% RSLogix 500 project wind.RSS %
PROJECT "WIND"    % processor: SLC 500, 1747-L543 %

PROGRAM FILES
  LAD 2 "MAIN"  12 rungs  %   %
  LAD 3 "AZ MAN CON"  4 rungs
  LAD 4 "AZ PID CON"  7 rungs
  LAD 5 "DATA XFER"  3 rungs
  LAD 6 "ALT MAN C"  4 rungs
  LAD 7 "ALT PID C"  6 rungs

DATA FILES
  O0 OUTPUT  21 elements
  I1 INPUT  21 elements
  S2 STATUS  164 elements
  B3 BINARY  1 elements
  T4 TIMER  1 elements
  C5 COUNTER  1 elements
  R6 CONTROL  1 elements
  N7 INTEGER  30 elements
  F8 FLOAT  1 elements
  N10 AZ PID  30 elements  % PID Control File %
  N11 ALT PID  30 elements

LADDER 2 "MAIN"    %   %
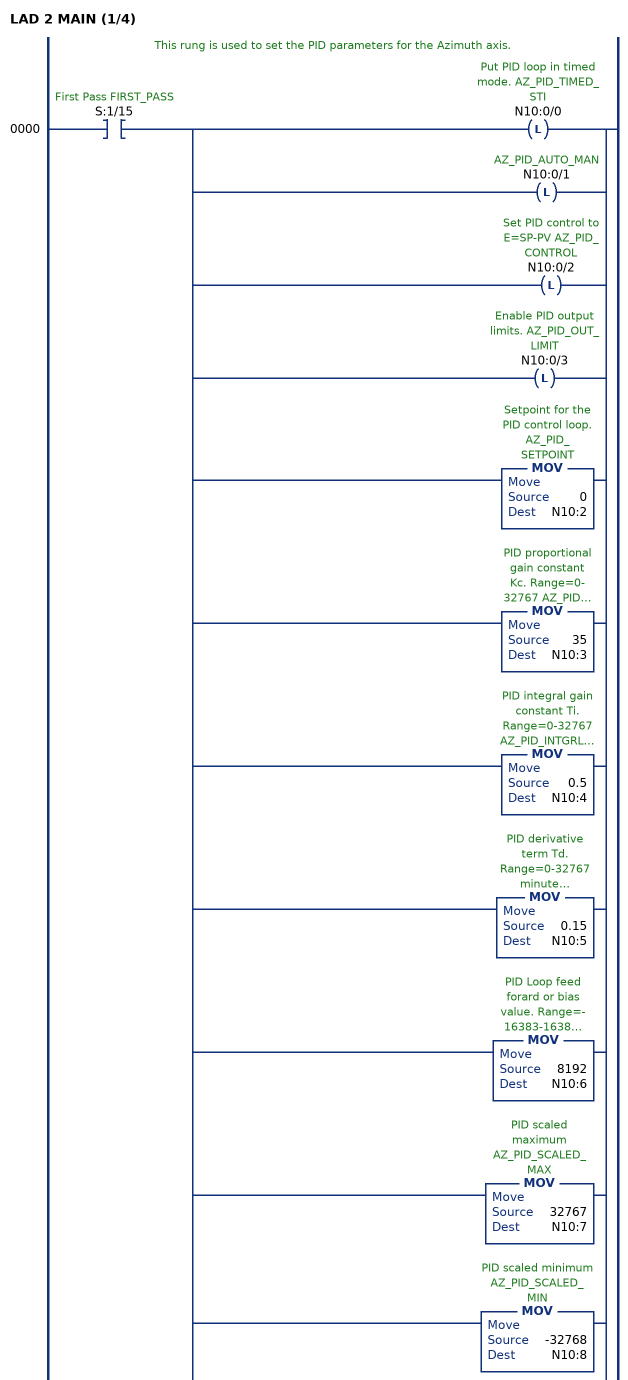
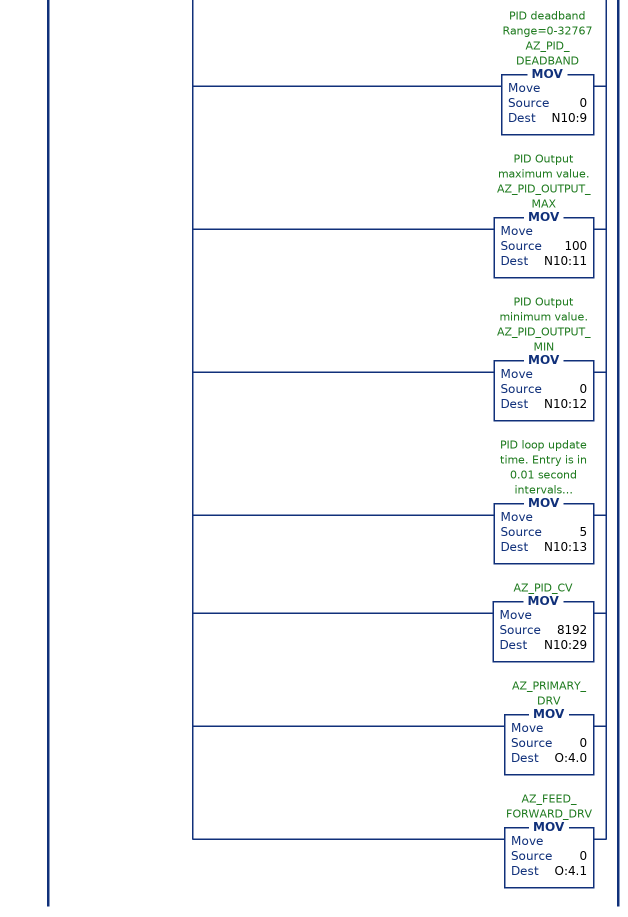
% Rung: 0 %
% This rung is used to set the PID parameters for the Azimuth axis. %
SOR XIC S:1/15 BST OTL N10:0/0 NXB OTL N10:0/1 NXB OTL N10:0/2 NXB OTL N10:0/3 NXB MOV 0 N10:2 NXB MOV 35 N10:3 NXB MOV 0.5 N10:4 NXB MOV 0.15 N10:5 NXB MOV 8192 N10:6 NXB MOV 32767 N10:7 NXB MOV -32768 N10:8 NXB MOV 0 N10:9 NXB MOV 100 N10:11 NXB MOV 0 N10:12 NXB MOV 5 N10:13 NXB MOV 8192 N10:29 NXB MOV 0 O:4.0 NXB MOV 0 O:4.1 BND EOR
%   S:1/15  FIRST_PASS  "First Pass" %
%   N10:0/0  AZ_PID_TIMED_STI  "Put PID loop in timed mode." %
%   N10:0/1  AZ_PID_AUTO_MAN %
%   OTL N10:0/1  "Put PID Loop in Manual Control." %
%   N10:0/2  AZ_PID_CONTROL  "Set PID control to E=SP-PV" %
%   N10:0/3  AZ_PID_OUT_LIMIT  "Enable PID output limits." %
%   N10:2  AZ_PID_SETPOINT  "Setpoint for the PID control loop." %
%   N10:3  AZ_PID_GAIN  "PID proportional gain constant Kc. Range=0-32767" %
%   N10:4  AZ_PID_INTGRL_GAIN  "PID integral gain constant Ti. Range=0-32767" %
%   N10:5  AZ_PID_DER_TERM  "PID derivative term Td. Range=0-32767 minutes" %
%   N10:6  AZ_PID_BIAS  "PID Loop feed forard or bias value. Range=-16383-16383" %
%   N10:7  AZ_PID_SCALED_MAX  "PID scaled maximum" %
%   N10:8  AZ_PID_SCALED_MIN  "PID scaled minimum" %
%   N10:9  AZ_PID_DEADBAND  "PID deadband Range=0-32767" %
%   N10:11  AZ_PID_OUTPUT_MAX  "PID Output maximum value." %
%   N10:12  AZ_PID_OUTPUT_MIN  "PID Output minimum value." %
%   N10:13  AZ_PID_LOOP_UPDATE  "PID loop update time. Entry is in 0.01 second intervals. Range=0.01-10.24 sec" %
%   N10:29  AZ_PID_CV %
%   O:4.0  AZ_PRIMARY_DRV %
%   MOV O:4.0  "Set Az Primary Control Output to zero." %
%   O:4.1  AZ_FEED_FORWARD_DRV %
%   MOV O:4.1  "Set Az feed forward output to zero." %

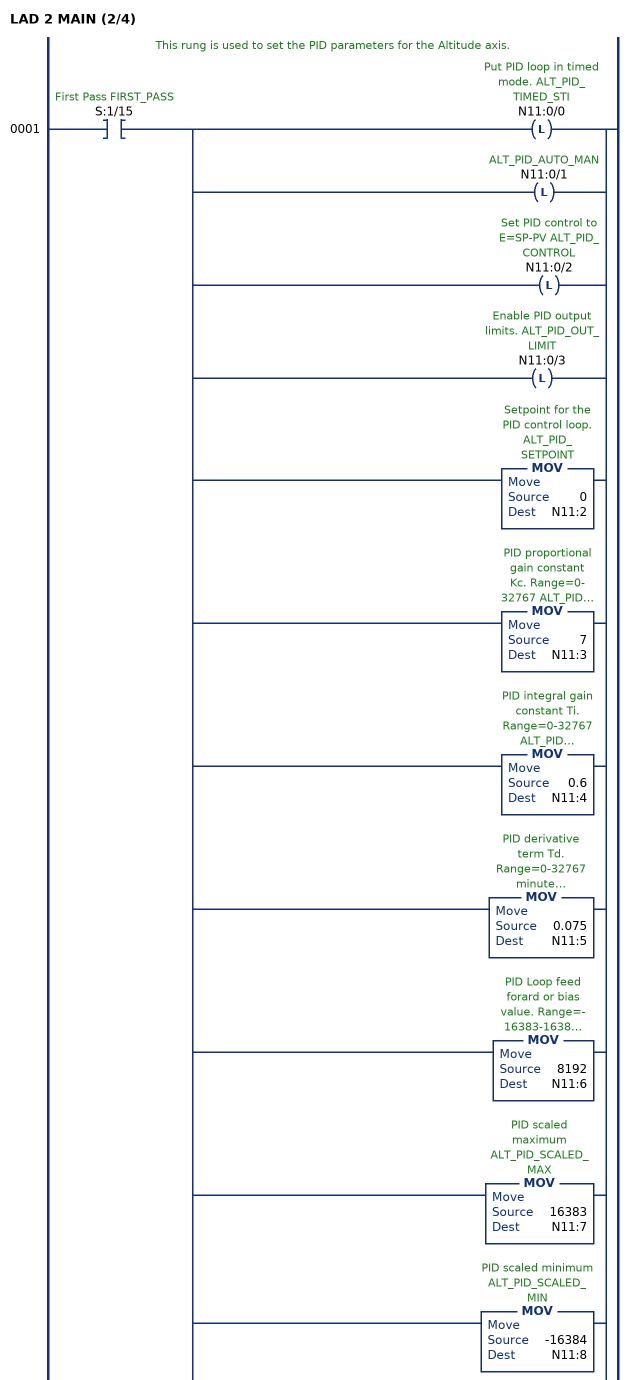

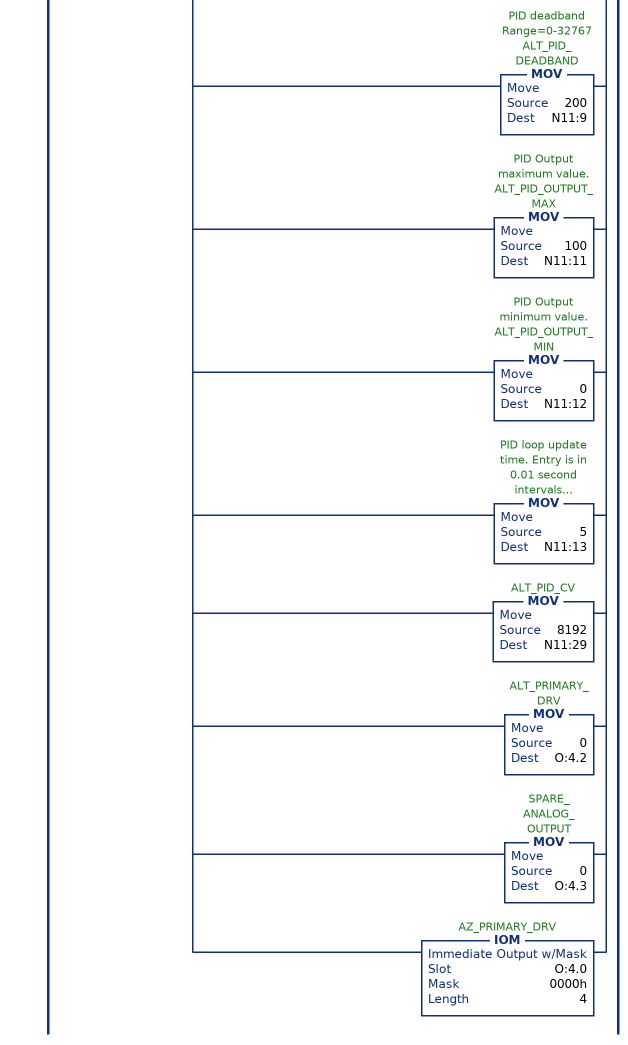
% Rung: 1 %
% This rung is used to set the PID parameters for the Altitude axis. %
SOR XIC S:1/15 BST OTL N11:0/0 NXB OTL N11:0/1 NXB OTL N11:0/2 NXB OTL N11:0/3 NXB MOV 0 N11:2 NXB MOV 7 N11:3 NXB MOV 0.6 N11:4 NXB MOV 0.075 N11:5 NXB MOV 8192 N11:6 NXB MOV 16383 N11:7 NXB MOV -16384 N11:8 NXB MOV 200 N11:9 NXB MOV 100 N11:11 NXB MOV 0 N11:12 NXB MOV 5 N11:13 NXB MOV 8192 N11:29 NXB MOV 0 O:4.2 NXB MOV 0 O:4.3 NXB IOM O:4.0 0000h 4 BND EOR
%   S:1/15  FIRST_PASS  "First Pass" %
%   N11:0/0  ALT_PID_TIMED_STI  "Put PID loop in timed mode." %
%   N11:0/1  ALT_PID_AUTO_MAN %
%   N11:0/2  ALT_PID_CONTROL  "Set PID control to E=SP-PV" %
%   N11:0/3  ALT_PID_OUT_LIMIT  "Enable PID output limits." %
%   N11:2  ALT_PID_SETPOINT  "Setpoint for the PID control loop." %
%   N11:3  ALT_PID_GAIN  "PID proportional gain constant Kc. Range=0-32767" %
%   N11:4  ALT_PID_INTGRL_GAIN  "PID integral gain constant Ti. Range=0-32767" %
%   N11:5  ALT_PID_DER_TERM  "PID derivative term Td. Range=0-32767 minutes" %
%   N11:6  ALT_PID_BIAS  "PID Loop feed forard or bias value. Range=-16383-16383" %
%   N11:7  ALT_PID_SCALED_MAX  "PID scaled maximum" %
%   N11:8  ALT_PID_SCALED_MIN  "PID scaled minimum" %
%   N11:9  ALT_PID_DEADBAND  "PID deadband Range=0-32767" %
%   N11:11  ALT_PID_OUTPUT_MAX  "PID Output maximum value." %
%   N11:12  ALT_PID_OUTPUT_MIN  "PID Output minimum value." %
%   N11:13  ALT_PID_LOOP_UPDATE  "PID loop update time. Entry is in 0.01 second intervals. Range=0.01-10.24 sec" %
%   N11:29  ALT_PID_CV %
%   O:4.2  ALT_PRIMARY_DRV %
%   MOV O:4.2  "Set Alt Primary Control Output to Zero." %
%   O:4.3  SPARE_ANALOG_OUTPUT %
%   O:4.0  AZ_PRIMARY_DRV %
%   IOM O:4.0  "Set output values immediatly." %

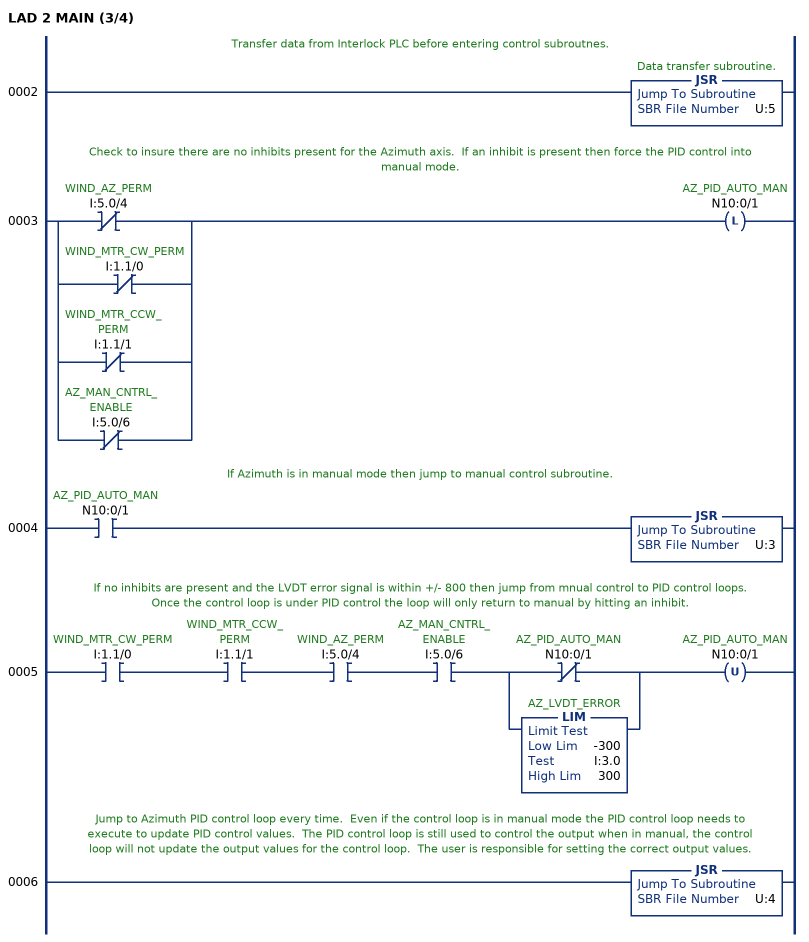
% Rung: 2 %
% Transfer data from Interlock PLC before entering control subroutnes. %
SOR JSR U:5 EOR
%   U:5  "Data transfer subroutine." %
% Rung: 3 %
% Check to insure there are no inhibits present for the Azimuth axis.  If an inhibit is present then force the PID control into manual mode. %
SOR BST XIO I:5.0/4 NXB XIO I:1.1/0 NXB XIO I:1.1/1 NXB XIO I:5.0/6 BND OTL N10:0/1 EOR
%   I:5.0/4  WIND_AZ_PERM %
%   I:1.1/0  WIND_MTR_CW_PERM %
%   I:1.1/1  WIND_MTR_CCW_PERM %
%   I:5.0/6  AZ_MAN_CNTRL_ENABLE %
%   N10:0/1  AZ_PID_AUTO_MAN %
%   OTL N10:0/1  "Put PID Loop in Manual Control." %
% Rung: 4 %
% If Azimuth is in manual mode then jump to manual control subroutine. %
SOR XIC N10:0/1 JSR U:3 EOR
%   N10:0/1  AZ_PID_AUTO_MAN %
%   JSR U:3  "JSR Az Manual Control Subroutine." %
% Rung: 5 %
% If no inhibits are present and the LVDT error signal is within +/- 800 then jump from mnual control to PID control loops.  Once the control loop is under PID control the loop will only return to manual by hitting an inhibit. %
SOR XIC I:1.1/0 XIC I:1.1/1 XIC I:5.0/4 XIC I:5.0/6 BST XIO N10:0/1 NXB LIM -300 I:3.0 300 BND OTU N10:0/1 EOR
%   I:1.1/0  WIND_MTR_CW_PERM %
%   I:1.1/1  WIND_MTR_CCW_PERM %
%   I:5.0/4  WIND_AZ_PERM %
%   I:5.0/6  AZ_MAN_CNTRL_ENABLE %
%   N10:0/1  AZ_PID_AUTO_MAN %
%   I:3.0  AZ_LVDT_ERROR %
% Rung: 6 %
% Jump to Azimuth PID control loop every time.  Even if the control loop is in manual mode the PID control loop needs to execute to update PID control values.  The PID control loop is still used to control the output when in manual, the control loop will not update the output values for the control loop.  The user is responsible for setting the correct output values. %
SOR JSR U:4 EOR
%   JSR U:4  "JSR Az PID Control Subroutine." %

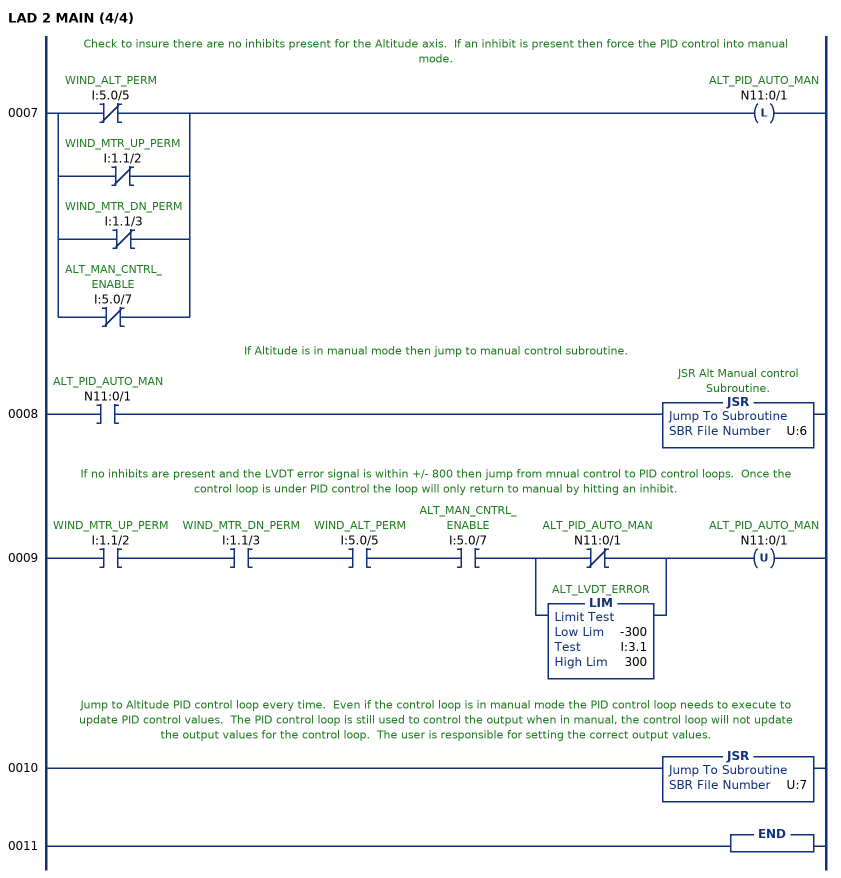
% Rung: 7 %
% Check to insure there are no inhibits present for the Altitude axis.  If an inhibit is present then force the PID control into manual mode. %
SOR BST XIO I:5.0/5 NXB XIO I:1.1/2 NXB XIO I:1.1/3 NXB XIO I:5.0/7 BND OTL N11:0/1 EOR
%   I:5.0/5  WIND_ALT_PERM %
%   I:1.1/2  WIND_MTR_UP_PERM %
%   I:1.1/3  WIND_MTR_DN_PERM %
%   I:5.0/7  ALT_MAN_CNTRL_ENABLE %
%   N11:0/1  ALT_PID_AUTO_MAN %
% Rung: 8 %
% If Altitude is in manual mode then jump to manual control subroutine. %
SOR XIC N11:0/1 JSR U:6 EOR
%   N11:0/1  ALT_PID_AUTO_MAN %
%   U:6  "JSR Alt Manual control Subroutine." %
% Rung: 9 %
% If no inhibits are present and the LVDT error signal is within +/- 800 then jump from mnual control to PID control loops.  Once the control loop is under PID control the loop will only return to manual by hitting an inhibit. %
SOR XIC I:1.1/2 XIC I:1.1/3 XIC I:5.0/5 XIC I:5.0/7 BST XIO N11:0/1 NXB LIM -300 I:3.1 300 BND OTU N11:0/1 EOR
%   I:1.1/2  WIND_MTR_UP_PERM %
%   I:1.1/3  WIND_MTR_DN_PERM %
%   I:5.0/5  WIND_ALT_PERM %
%   I:5.0/7  ALT_MAN_CNTRL_ENABLE %
%   N11:0/1  ALT_PID_AUTO_MAN %
%   I:3.1  ALT_LVDT_ERROR %
% Rung: 10 %
% Jump to Altitude PID control loop every time.  Even if the control loop is in manual mode the PID control loop needs to execute to update PID control values.  The PID control loop is still used to control the output when in manual, the control loop will not update the output values for the control loop.  The user is responsible for setting the correct output values. %
SOR JSR U:7 EOR
%   JSR U:7  "JSR Alt PID control subroutine." %
% Rung: 11 %
SOR END EOR

LADDER 3 "AZ MAN CON"
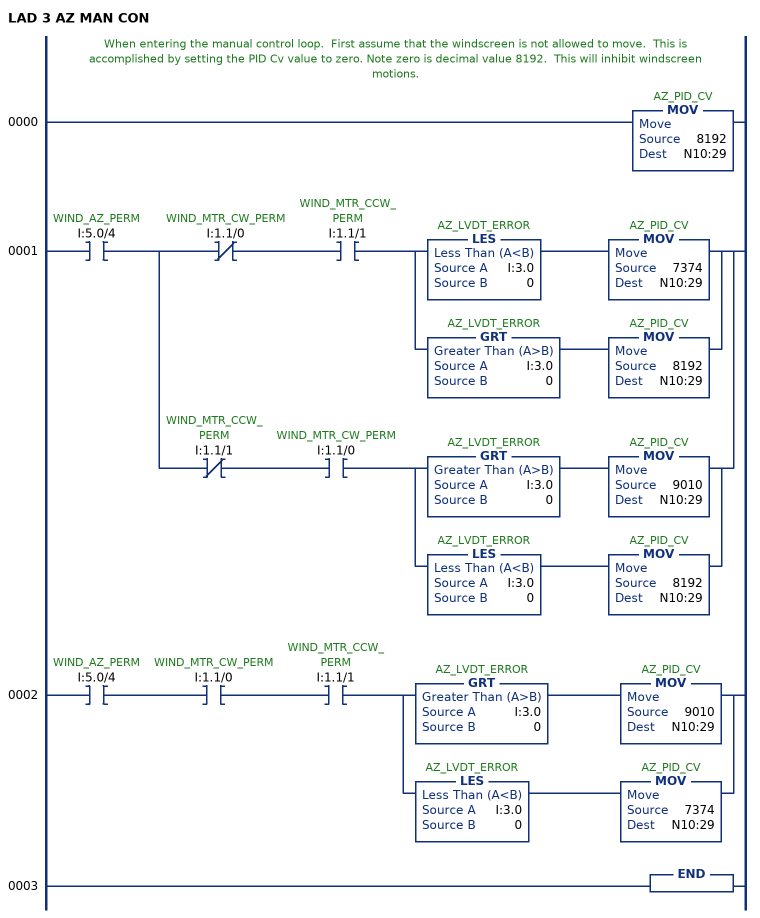
% Rung: 0 %
% When entering the manual control loop.  First assume that the windscreen is not allowed to move.  This is accomplished by setting the PID Cv value to zero. Note zero is decimal value 8192.  This will inhibit windscreen motions. %
SOR MOV 8192 N10:29 EOR
%   N10:29  AZ_PID_CV %
% Rung: 1 %
SOR XIC I:5.0/4 BST XIO I:1.1/0 XIC I:1.1/1 BST LES I:3.0 0 MOV 7374 N10:29 NXB GRT I:3.0 0 MOV 8192 N10:29 BND NXB XIO I:1.1/1 XIC I:1.1/0 BST GRT I:3.0 0 MOV 9010 N10:29 NXB LES I:3.0 0 MOV 8192 N10:29 BND BND EOR
%   I:5.0/4  WIND_AZ_PERM %
%   I:1.1/0  WIND_MTR_CW_PERM %
%   I:1.1/1  WIND_MTR_CCW_PERM %
%   I:3.0  AZ_LVDT_ERROR %
%   N10:29  AZ_PID_CV %
% Rung: 2 %
SOR XIC I:5.0/4 XIC I:1.1/0 XIC I:1.1/1 BST GRT I:3.0 0 MOV 9010 N10:29 NXB LES I:3.0 0 MOV 7374 N10:29 BND EOR
%   I:5.0/4  WIND_AZ_PERM %
%   I:1.1/0  WIND_MTR_CW_PERM %
%   I:1.1/1  WIND_MTR_CCW_PERM %
%   I:3.0  AZ_LVDT_ERROR %
%   N10:29  AZ_PID_CV %
% Rung: 3 %
SOR END EOR

LADDER 4 "AZ PID CON"
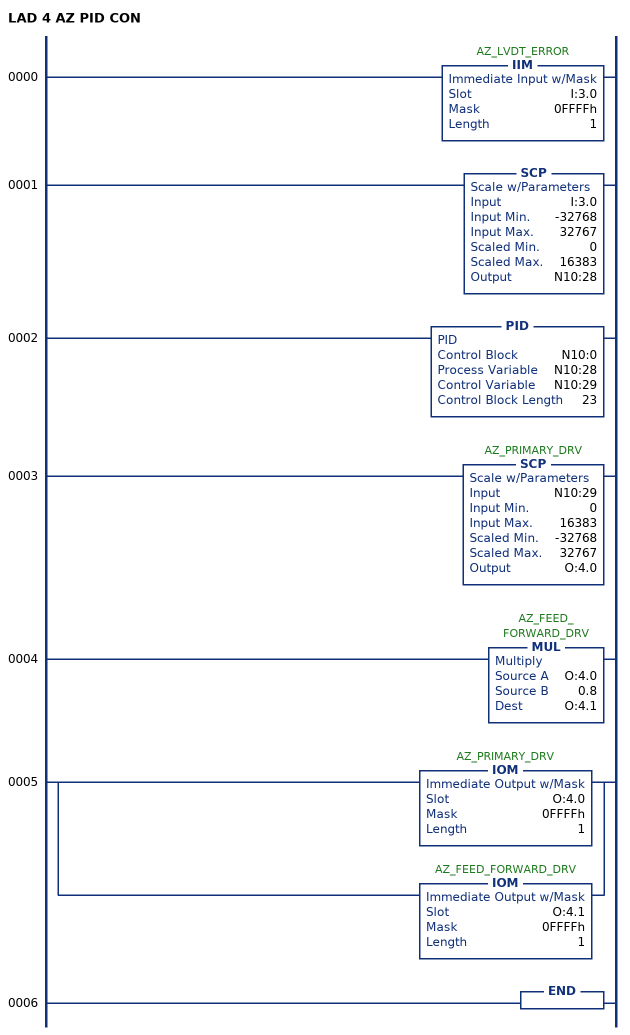
% Rung: 0 %
SOR IIM I:3.0 0FFFFh 1 EOR
%   I:3.0  AZ_LVDT_ERROR %
% Rung: 1 %
SOR SCP I:3.0 -32768 32767 0 16383 N10:28 EOR
%   I:3.0  AZ_LVDT_ERROR %
% Rung: 2 %
SOR PID N10:0 N10:28 N10:29 23 EOR
%   N10:29  AZ_PID_CV %
% Rung: 3 %
SOR SCP N10:29 0 16383 -32768 32767 O:4.0 EOR
%   N10:29  AZ_PID_CV %
%   O:4.0  AZ_PRIMARY_DRV %
% Rung: 4 %
SOR MUL O:4.0 0.8 O:4.1 EOR
%   O:4.0  AZ_PRIMARY_DRV %
%   O:4.1  AZ_FEED_FORWARD_DRV %
% Rung: 5 %
SOR BST IOM O:4.0 0FFFFh 1 NXB IOM O:4.1 0FFFFh 1 BND EOR
%   O:4.0  AZ_PRIMARY_DRV %
%   IOM O:4.0  "Set output values immediatly." %
%   O:4.1  AZ_FEED_FORWARD_DRV %
% Rung: 6 %
SOR END EOR

LADDER 5 "DATA XFER"
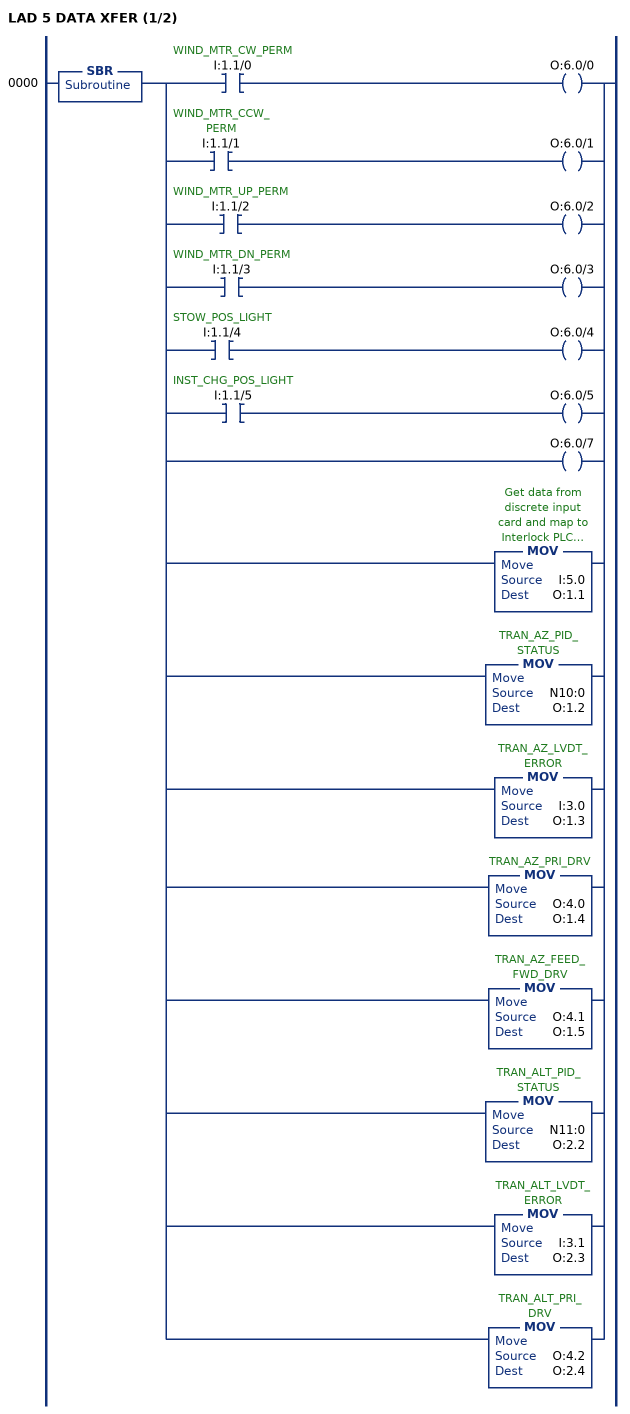
% Rung: 0 %
SOR SBR BST XIC I:1.1/0 OTE O:6.0/0 NXB XIC I:1.1/1 OTE O:6.0/1 NXB XIC I:1.1/2 OTE O:6.0/2 NXB XIC I:1.1/3 OTE O:6.0/3 NXB XIC I:1.1/4 OTE O:6.0/4 NXB XIC I:1.1/5 OTE O:6.0/5 NXB OTE O:6.0/7 NXB MOV I:5.0 O:1.1 NXB MOV N10:0 O:1.2 NXB MOV I:3.0 O:1.3 NXB MOV O:4.0 O:1.4 NXB MOV O:4.1 O:1.5 NXB MOV N11:0 O:2.2 NXB MOV I:3.1 O:2.3 NXB MOV O:4.2 O:2.4 BND EOR
%   I:1.1/0  WIND_MTR_CW_PERM %
%   I:1.1/1  WIND_MTR_CCW_PERM %
%   I:1.1/2  WIND_MTR_UP_PERM %
%   I:1.1/3  WIND_MTR_DN_PERM %
%   I:1.1/4  STOW_POS_LIGHT %
%   I:1.1/5  INST_CHG_POS_LIGHT %
%   I:5.0  DC_INPUT_MODULE %
%   O:1.1  TRAN_DC_INPUT_MODULE  "Get data from discrete input card and map to Interlock PLC." %
%   O:1.2  TRAN_AZ_PID_STATUS %
%   I:3.0  AZ_LVDT_ERROR %
%   O:1.3  TRAN_AZ_LVDT_ERROR %
%   O:4.0  AZ_PRIMARY_DRV %
%   MOV O:4.0  "Set Az Primary Control Output to zero." %
%   O:1.4  TRAN_AZ_PRI_DRV %
%   O:4.1  AZ_FEED_FORWARD_DRV %
%   MOV O:4.1  "Set Az feed forward output to zero." %
%   O:1.5  TRAN_AZ_FEED_FWD_DRV %
%   O:2.2  TRAN_ALT_PID_STATUS %
%   I:3.1  ALT_LVDT_ERROR %
%   O:2.3  TRAN_ALT_LVDT_ERROR %
%   O:4.2  ALT_PRIMARY_DRV %
%   MOV O:4.2  "Set Alt Primary Control Output to Zero." %
%   O:2.4  TRAN_ALT_PRI_DRV %

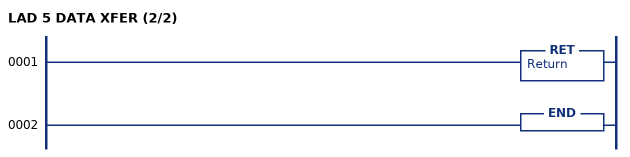
% Rung: 1 %
SOR RET EOR
% Rung: 2 %
SOR END EOR

LADDER 6 "ALT MAN C"
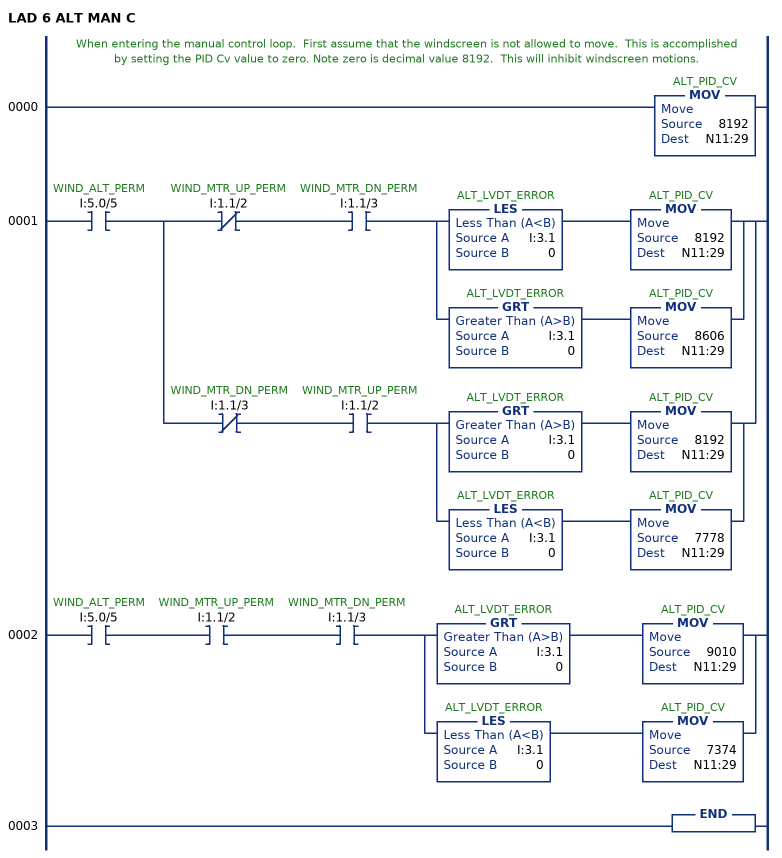
% Rung: 0 %
% When entering the manual control loop.  First assume that the windscreen is not allowed to move.  This is accomplished by setting the PID Cv value to zero. Note zero is decimal value 8192.  This will inhibit windscreen motions. %
SOR MOV 8192 N11:29 EOR
%   N11:29  ALT_PID_CV %
% Rung: 1 %
SOR XIC I:5.0/5 BST XIO I:1.1/2 XIC I:1.1/3 BST LES I:3.1 0 MOV 8192 N11:29 NXB GRT I:3.1 0 MOV 8606 N11:29 BND NXB XIO I:1.1/3 XIC I:1.1/2 BST GRT I:3.1 0 MOV 8192 N11:29 NXB LES I:3.1 0 MOV 7778 N11:29 BND BND EOR
%   I:5.0/5  WIND_ALT_PERM %
%   I:1.1/2  WIND_MTR_UP_PERM %
%   I:1.1/3  WIND_MTR_DN_PERM %
%   I:3.1  ALT_LVDT_ERROR %
%   N11:29  ALT_PID_CV %
% Rung: 2 %
SOR XIC I:5.0/5 XIC I:1.1/2 XIC I:1.1/3 BST GRT I:3.1 0 MOV 9010 N11:29 NXB LES I:3.1 0 MOV 7374 N11:29 BND EOR
%   I:5.0/5  WIND_ALT_PERM %
%   I:1.1/2  WIND_MTR_UP_PERM %
%   I:1.1/3  WIND_MTR_DN_PERM %
%   I:3.1  ALT_LVDT_ERROR %
%   N11:29  ALT_PID_CV %
% Rung: 3 %
SOR END EOR

LADDER 7 "ALT PID C"
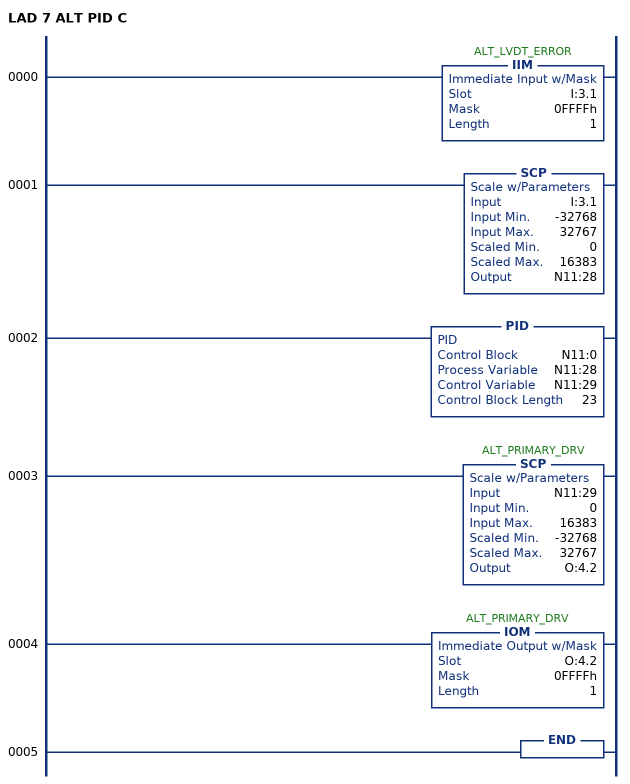
% Rung: 0 %
SOR IIM I:3.1 0FFFFh 1 EOR
%   I:3.1  ALT_LVDT_ERROR %
% Rung: 1 %
SOR SCP I:3.1 -32768 32767 0 16383 N11:28 EOR
%   I:3.1  ALT_LVDT_ERROR %
% Rung: 2 %
SOR PID N11:0 N11:28 N11:29 23 EOR
%   N11:29  ALT_PID_CV %
% Rung: 3 %
SOR SCP N11:29 0 16383 -32768 32767 O:4.2 EOR
%   N11:29  ALT_PID_CV %
%   O:4.2  ALT_PRIMARY_DRV %
% Rung: 4 %
SOR IOM O:4.2 0FFFFh 1 EOR
%   O:4.2  ALT_PRIMARY_DRV %
% Rung: 5 %
SOR END EOR

OTHER DOCUMENTED ADDRESSES
  DFILE:0  "OUTPUT"
  DFILE:1  "INPUT"
  DFILE:2  "STATUS"
  DFILE:3  "BINARY"
  DFILE:4  "TIMER"
  DFILE:5  "COUNTER"
  DFILE:6  "CONTROL"
  DFILE:7  "INTEGER"
  DFILE:8  "FLOAT"
  DFILE:9  "ALT PID"
  DFILE:10  "AZ PID PID Control File"
  DFILE:11  "ALT PID"
  I:1.0  INTLK_PLC_COM_STATUS
  I:5.0/0  WIND_AZ1_FLT
  I:5.0/1  WIND_AZ2_FLT
  I:5.0/2  WIND_AZ3_FLT
  I:5.0/3  WIND_ALT1_FLT
  I:5.0/15  LOW_LVL_LIGHTING_REQ
  O:1.0  DCM_COM_STATUS
  O:1.1/0  TRAN_WIND_AZ1_FLT
  O:1.1/1  TRAN_WIND_AZ2_FLT
  O:1.1/2  TRAN_WIND_AZ3_FLT
  O:1.1/3  TRAN_WIND_ALT1_FLT
  O:1.1/4  TRAN_WIND_AZ_PERM
  O:1.1/5  TRAN_WIND_ALT_PERM
  O:9.0  RELAY_OUTPUT_MODULE

OTHER INSTRUCTION COMMENTS
  O:9.0 MOV  "Get data from Interlock PLC and map to relay output card."

REVISION NOTES
  2: added Az Pid Control
  32: Initial release for the SDSS telescope windscreen controls.
  71: First revision to add alt control
  73: changed alt pid gain destination
  75: AZ PID Gain 30
     AZ PID Deadband 400
  82: Changed Alt maximum scaled output from 32763 to 16383 and -32764 to -16384
  103: swapped slow approach directions
  104: swapped directions for slow approach inside loops

DATA TABLE (non-zero values as saved)
DATA N10
% N10:0 % -24547 0 0 35 1 0 8192 32767 -32768 0
% N10:10 % 0 100 0 5 -3 -3 50 13 10946 1
% N10:20 % -16 11850 0 0 0 0 0 0 8191 8205
DATA N11
% N11:0 % -24305 0 0 7 1 0 8192 16383 -16384 200
% N11:10 % 0 100 0 5 14 14 50 0 20228 2
% N11:20 % 112 12012 0 0 0 0 0 0 8199 8192
